// SIMATIC S7-200 project (STEP 7-Micro/WIN), CPU 221 REL 01.10

SYMBOL_TABLE USER1
CB               Q0.0     // chuong bao
END_SYMBOL_TABLE

ORGANIZATION_BLOCK MAIN:OB1
TITLE=PROGRAM COMMENTS
BEGIN
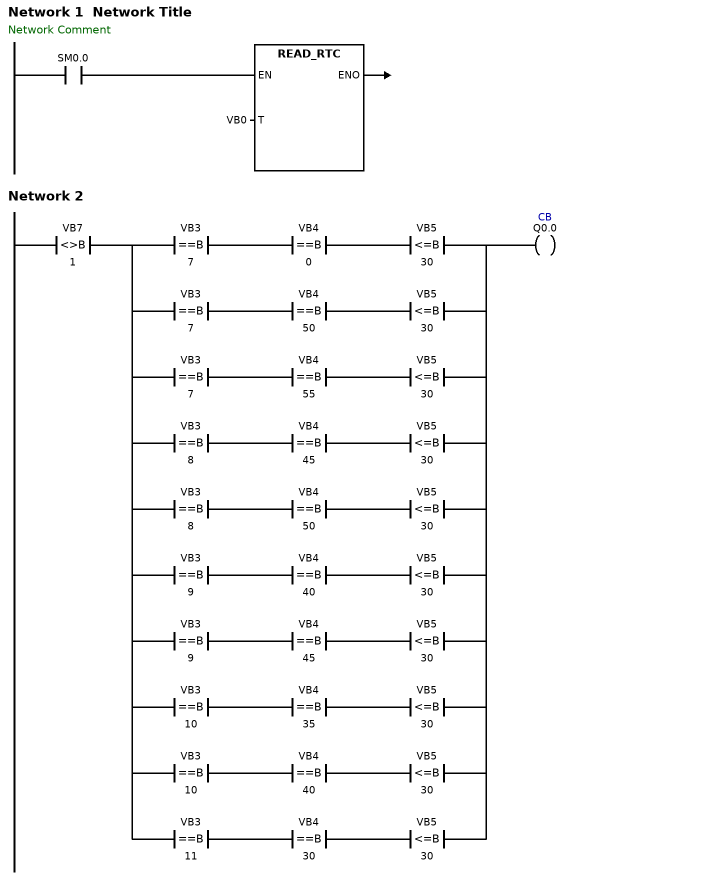
Network 1 // Network Title
// Network Comment
LD     SM0.0
TODR   VB0
Network 2
LDB<>  VB7, 1
LDB=   VB3, 7
AB=    VB4, 0
AB<=   VB5, 30
LDB=   VB3, 7
AB=    VB4, 50
AB<=   VB5, 30
OLD
LDB=   VB3, 7
AB=    VB4, 55
AB<=   VB5, 30
OLD
LDB=   VB3, 8
AB=    VB4, 45
AB<=   VB5, 30
OLD
LDB=   VB3, 8
AB=    VB4, 50
AB<=   VB5, 30
OLD
LDB=   VB3, 9
AB=    VB4, 40
AB<=   VB5, 30
OLD
LDB=   VB3, 9
AB=    VB4, 45
AB<=   VB5, 30
OLD
LDB=   VB3, 10
AB=    VB4, 35
AB<=   VB5, 30
OLD
LDB=   VB3, 10
AB=    VB4, 40
AB<=   VB5, 30
OLD
LDB=   VB3, 11
AB=    VB4, 30
AB<=   VB5, 30
OLD
ALD
=      CB:Q0.0
END_ORGANIZATION_BLOCK
